// TIA Portal V18 export
FUNCTION "DOvar" : Void   // FC10010, LAD
{ S7_Optimized_Access := 'TRUE' }
VERSION : 0.1
// stored: AutoNumber false, IsIECCheckEnabled false, SetENOAutomatically false, UDAEnableTagReadback false
   VAR_INPUT
      iFuncSystem : Byte;
      iFuncVar : Byte;
   END_VAR
   VAR_OUTPUT
      xOutput : Bool;
   END_VAR
BEGIN

REGION Network 1 (SCL)
   CASE #iFuncSystem OF
       0:  // Statement section case 2 to 4
           ;
       1..3:  // Statement section case 1
           CASE #iFuncVar OF
               0:  // 
                   ;
               1:  // 
                   #xOutput := "AHUDO".Requests.xHeaterPumpCmd[#iFuncSystem];
               2:  // 
                   #xOutput := "AHUDO".Requests.xSAFAnalogEnable[#iFuncSystem];
               3:  // 
                   #xOutput := "AHUDO".Requests.xSAFSp1Cmd[#iFuncSystem];
               4:  // 
                   #xOutput := "AHUDO".Requests.xSAFSp2Cmd[#iFuncSystem];
           END_CASE;
        4..9:
            ;
        10:
            CASE #iFuncVar OF
                0:  // 
                    ;
                1:  // 
                    #xOutput := "HCsDO".Requests.xHC3wvIncrease[1];
                2:  // 
                    #xOutput := "HCsDO".Requests.xHC3wvDecrease[1];
                3:  // 
                    #xOutput := "HCsDO".Requests.xHC3wvIncrease[2];
                4:  // 
                    #xOutput := "HCsDO".Requests.xHC3wvDecrease[2];
                5:  //
                    #xOutput := "HCsDO".Requests.xHCPump1Cmd[1];
                6:  //
                    #xOutput := "HCsDO".Requests.xHCPump2Cmd[1];
                7:  //
                    #xOutput := "HCsDO".Requests.xHCPump1Cmd[2];
                8:  //
                    #xOutput := "HCsDO".Requests.xHCPump2Cmd[2];
                9:  //    
                    ;
                10:
                    #xOutput := "HSsDO".Requests.xBoilerEnable[1];
                11:
                    #xOutput := "HSsDO".Requests.xBoilerSt1Enable[1];
                12:
                    #xOutput := "HSsDO".Requests.xBoilerSt2Enable[1];
                13:
                    #xOutput := "HSsDO".Requests.xBoilerShuntPumpEnable[1];
                14:
                    #xOutput := "HSsDO".Requests.xBoilerShutOffValveCmd[1];
                15:
                    ;
                16:
                    #xOutput := "HSsDO".Requests.xBoilerEnable[2];
                17:
                    #xOutput := "HSsDO".Requests.xBoilerSt1Enable[2];
                18:
                    #xOutput := "HSsDO".Requests.xBoilerSt2Enable[2];
                19:
                    #xOutput := "HSsDO".Requests.xBoilerShuntPumpEnable[2];
                20:
                    #xOutput := "HSsDO".Requests.xBoilerShutOffValveCmd[2];
                ELSE:
                    ;
            END_CASE;
        11..99:
            ;
        100:    //DieselLine
            CASE #iFuncVar OF
                0:  // 
                    ;
                1:  // 
                    #xOutput := "DLsDO".Requests.xDieselLineHeatingCmd[1];
                2:  // 
                    #xOutput := "DLsDO".Requests.xDieselLineHeatingCmd[2];
                3:  // 
                    #xOutput := "DLsDO".Requests.xDieselLinePumpEnable;
                4:  // 
                    #xOutput := "DLsDO".Requests.xDieselLinePumpSelect;
                5:  //
                    #xOutput := "DLsDO".Requests.xDieselLineDayTankValve[1];
                6:  //
                    #xOutput := "DLsDO".Requests.xDieselLineDayTankValve[2];
                ELSE:
                    ;
            END_CASE;
       ELSE  // Statement section ELSE
           ;
   END_CASE;
END_REGION
END_FUNCTION
